{attribute 'qualified_only'}
{attribute 'strict'}
TYPE ePeakshaveMode :
(
	Multiphase := 0,
	Singlephase := 1
);
END_TYPE

(* stored: Version 1.1.0.1, ProductVersion 3.1.4026.18
   DUT ePeakshaveMode: Id {23e48150-7e39-4fae-9c89-db74ed0bd99d} *)
